PROGRAM MAIN
VAR
	j_digitalInput1 AT%I*:BOOL;
END_VAR

END_PROGRAM

(* stored: Version 1.1.0.1, ProductVersion 3.1.4024.2
   POU MAIN: Id {60dfe297-14aa-41d4-bcd0-9ac131306f78}, SpecialFunc None *)
